// TIA Portal V16 export
// export: Created 2024-12-03T15:41:40.7608411Z, ExportSetting WithDefaults, DisplayName Totally Integrated Automation Portal, DisplayVersion V16 Update 6, DisplayName TIA Portal Version Control Interface, DisplayVersion V16 Update 2, DisplayName TIA Portal Openness, DisplayVersion V16 Update 6, DisplayName TIA Portal Teamcenter Gateway, DisplayVersion V16, DisplayName SINAMICS Startdrive Advanced, DisplayVersion V16 Update 5, DisplayName SINAMICS Startdrive G130, G150, S120, S150, SINAMICS MV, S210, DisplayVersion V16 Update 5, DisplayName SINAMICS Startdrive G110M, G120, G120C, G120D, G120P, G115D, DisplayVersion V16 Update 5, DisplayName STEP 7 Professional, DisplayVersion V16 Update 6, DisplayName STEP 7 Safety, DisplayVersion V16, DisplayName WinCC Advanced / Unified PC, DisplayVersion V16 Update 6
FUNCTION_BLOCK "HMI_Main_FB"   // FB55, SCL
{ S7_Optimized_Access := 'TRUE' }
VERSION : 0.1
// stored: AutoNumber true, IsIECCheckEnabled false, IsRetainMemResEnabled false, MemoryReserve 100, SetENOAutomatically false, UDAEnableTagReadback false
BEGIN
   REGION Reload settings

       IF "FirstScan" THEN
           "HMI_DB".ReloadSettings.signal := 1;
       END_IF;



       "Util_HandShaked_FC"(IO_Shake := "HMI_DB".ReloadSettings);
       "Util_HandShaked_FC"(IO_Shake := "HMI_DB".RemoveManualOverride);
       "Util_HandShaked_FC"(IO_Shake :=  "HMI_DB".ResetCounters);
       "Util_HandShaked_FC"(IO_Shake :=  "HMI_DB".SetDefaultTrackings);
       "Util_HandShaked_FC"(IO_Shake := "HMI_DB".ResetSensorCounters);

   END_REGION
END_FUNCTION_BLOCK
